KUKA KRL data list: fFrame.dat

&ACCESS RV1
&REL 2
DEFDAT  fframe PUBLIC


DECL GLOBAL FRAME gfBaseShift[6]
gfBaseShift[1]={X -5.00000,Y -5.00000,Z 0.00000,A 0.0,B 0.0,C 0.0}
gfBaseShift[2]={X -16,Y -16.0000,Z 0.0,A 0.0,B 0.0,C 0.0}
gfBaseShift[3]={X 0.000,Y 0.0000,Z 0.0000,A 0.0,B 0.0,C 0.0}
gfBaseShift[4]={X 0.000,Y 0.0000,Z 0.0000,A 0.0,B 0.0,C 0.0}
gfBaseShift[5]={X 0.000,Y 0.0000,Z 0.0000,A 0.0,B 0.0,C 0.0}
gfBaseShift[6]={X -16,Y -16.0000,Z 0.0,A 0.0,B 0.0,C 0.0}
ENDDAT
